TYPE ST_ProductHandlingProdPar :
STRUCT
	GantryA						: ST_GantryProdPar;
	GantryB						: ST_GantryProdPar;
	OutfeedConveyor				: ST_OutfeedConveyorProdPar;

END_STRUCT
END_TYPE

(* stored: Version 1.1.0.1, ProductVersion 3.1.4020.12
   DUT ST_ProductHandlingProdPar: Id {e74d7f13-f637-401c-a070-4731e595530d} *)
